INTERFACE I_MotionAxisNC EXTENDS I_MotionAxisCommon

(*
    Check all post condition before updating bCommandedMoveAbsolute
    The implmentatation will depend on the axis type
    DS402 NC/Direct axis : Implementation need to check that the drive is in the correct mode before initaiting the move then set bCommandedMoveAbsolute
    MP NC axis : will immediately write to bCommandedMoveAbsolute
*)
METHOD StartMove : BOOL
VAR_INPUT
	MoveMode	: E_EpicsMotorCmd;
	CmdExecute	: BOOL;
END_VAR
END_METHOD

END_INTERFACE

(* stored: Version 1.1.0.1
   Itf I_MotionAxisNC: Id {988e1537-42fa-4f3b-9835-b781579a345f}
   Method StartMove: Id {da366508-7b88-44b9-b101-027048fd2ba1} *)
